// TIA Portal V20 export
FUNCTION "FC_ResetPositionData" : Void   // FC700, SCL
{ S7_Optimized_Access := 'TRUE' }
// stored: AutoNumber false, SetENOAutomatically false
   VAR_INPUT
      iDataPosition : Int;   // Data Positions(1..5)
   END_VAR
   VAR_TEMP
      tIndex : Int;
   END_VAR
BEGIN
   REGION Description header 
       //==================================================================================
       // POSALUX Swiss SA / (C) Copyright 2025
       //----------------------------------------------------------------------------------
       // Title: FC_Fill_Data_Record
       // Comment/Function: Mise à jour des datas d'une pièce
       //
       // Author: Fabien Waldt
       // Engineering: TIA Portal v17
       //----------------------------------------------------------------------------------
       // Change log table:
       // Version  | Date     | Expert in charge | Changes applied
       // ---------|----------|------------------|------------------------------------
       // 00.00.01 | 20250224 | FWA              | First released version
       // ==================================================================================
   END_REGION
   "DB_DataPositions".Position[#iDataPosition].Part_id := 0;
       "DB_DataPositions".Position[#iDataPosition].Status := 0;
       "DB_DataPositions".Position[#iDataPosition].FailCode := 0;
       "DB_DataPositions".Position[#iDataPosition].FailCodeBackwall := 0;
       "DB_DataPositions".Position[#iDataPosition].WOZ_Status := 0;
       "DB_DataPositions".Position[#iDataPosition].WOC_Status := 0;
       "DB_DataPositions".Position[#iDataPosition].WOZ_Measure := 0.0;
       "DB_DataPositions".Position[#iDataPosition].WOC_Measure := 0;
       "DB_DataPositions".Position[#iDataPosition].TotalCycleTime := 0;
       "DB_DataPositions".Position[#iDataPosition].LaserCycleTime := 0;
       "DB_DataPositions".Position[#iDataPosition].MeasureLoadCycleTime := 0;
       FOR #tIndex := 19 TO 0 BY -1 DO
           "DB_DataPositions".Position[#iDataPosition].DMC[#tIndex] := 0;
       END_FOR;
       "DB_DataPositions".Position[#iDataPosition].OrderNbr := '---';
       "DB_DataPositions".Position[#iDataPosition].IdentNbr := '---';
       "DB_DataPositions".Position[#iDataPosition].BatchNbr := '---';
       "DB_DataPositions".Position[#iDataPosition].OperatorNbr := '---';
       "DB_DataPositions".Position[#iDataPosition].Comment := '---';
       FOR #tIndex := 0 TO 99 BY 1 DO
           "DB_DataPositions".Position[#iDataPosition].HoleSettings[#tIndex].Measure_X := 0;
           "DB_DataPositions".Position[#iDataPosition].HoleSettings[#tIndex].Measure_Y := 0;
           "DB_DataPositions".Position[#iDataPosition].HoleSettings[#tIndex].Measure_Z := 0;
           "DB_DataPositions".Position[#iDataPosition].HoleSettings[#tIndex].Measure_D := 0;
           "DB_DataPositions".Position[#iDataPosition].HoleSettings[#tIndex].Measure_Z := 0;
           "DB_DataPositions".Position[#iDataPosition].HoleSettings[#tIndex].Measure_concentricity_before := 0;
           "DB_DataPositions".Position[#iDataPosition].HoleSettings[#tIndex].Measure_concentricity_after := 0;
           "DB_DataPositions".Position[#iDataPosition].HoleSettings[#tIndex].Job_laser := 0;
       END_FOR;
END_FUNCTION
